{attribute 'GeneratedUsingTerminal: EL7037-0000-0016'}
{attribute addProperty BoxType "EL7037-0000-0016"}
{attribute addProperty Id "StatusAT %I*Status_1E008DB912"}
{attribute addProperty CRC "3725421367"}
{attribute addProperty Size "12"}
TYPE STM_Status_DE0D6B37 :
STRUCT
	{attribute addProperty Name "Status"}
	Status AT %I* : Status_1E008DB9;
END_STRUCT
END_TYPE

(* stored: Version 1.2.0.0, ProductVersion 3.1.4024.9
   DUT STM_Status_DE0D6B37: Id {bca5c3d1-e9c1-4ea7-8c21-5ce962eae998} *)
